FUNCTION_BLOCK FB_Example
VAR
    BeginTime : TIME;
END_VAR
BEGIN
BeginTime := T#5s;
END_FUNCTION_BLOCK
